FUNCTION_BLOCK FB_Girar_SFC

VAR_INPUT
    // SFC-Flags
    SFCPause: BOOL;
    SFCReset: BOOL;
    
    // Parametros de control de la estacion
    CicloACiclo: BOOL;    

	// Sincronizacion
    Benido: BOOL ;
    Ejecuta: BOOL;

    PlatoEmpujadorDetras AT %I* : BOOL;
END_VAR
VAR_OUTPUT
    //PlatoEmpujadorAvanza AT %Q* : BOOL;
   // PlatoRetenedorAtras AT %Q* : BOOL;
	PlatoEmpujadorAvanza: BOOL;
    PlatoRetenedorAtras: BOOL;
	// Sincronizacion    
    Acabhe: BOOL;
    ListoKalisto: BOOL;
END_VAR
VAR_IN_OUT
	Tapas : ARRAY[0..7] OF ST_POSICION;
    TapaAuxRot : ST_POSICION; 
END_VAR

VAR 
	i : UINT;
END_VAR

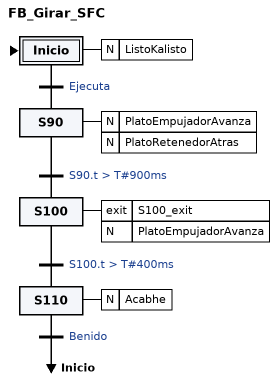
INITIAL_STEP Inicio:
    ListoKalisto(N);
END_STEP
TRANSITION FROM Inicio TO S90
    := Ejecuta;
END_TRANSITION
STEP S90:
    PlatoEmpujadorAvanza(N);
    PlatoRetenedorAtras(N);
END_STEP
TRANSITION FROM S90 TO S100
    := S90.t > T#900ms;
END_TRANSITION
STEP S100:
    S100_exit(P0);  // exit action
    PlatoEmpujadorAvanza(N);
END_STEP
TRANSITION FROM S100 TO S110
    := S100.t > T#400ms;
END_TRANSITION
STEP S110:
    Acabhe(N);
END_STEP
TRANSITION FROM S110 TO Inicio
    := Benido;
END_TRANSITION

ACTION RotArray:
TapaAuxRot := Tapas[7];

FOR i := 7 TO 1
 DO
 Tapas[i] := Tapas[i-1];	
END_FOR

Tapas[0] := TapaAuxRot;
END_ACTION

ACTION S100_exit:

END_ACTION

END_FUNCTION_BLOCK

(* stored: Version 1.1.0.1, ProductVersion 3.1.4024.12
   POU FB_Girar_SFC: Id {e2c5986b-0ebb-4426-b0b1-6207deec1967}, SpecialFunc None
   Action RotArray: Id {c4ed8f3e-9928-4c9c-bf72-ac50c896a4eb}
   Action S100_exit: Id {02c8a763-28f7-4fe9-ab00-f5cf9a6f4b28} *)
